// TIA Portal V20 export
TYPE "OPC_DestAssign"
// stored: Namespace ProductionLine
   STRUCT
      SourceSeq : Int;
      SourceNode : String[8];
      TotesID : String[10];
      WMSID : String[20];
      DestinationNode : String[8];
   END_STRUCT;
END_TYPE
